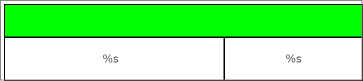
VISUALIZATION VISU_ETAPE_REGEN  // 363x81
VAR_IN_OUT
	COM: BLOCK_RS232_ONBOARD_V4;
END_VAR
    Textfield (4,37 220x44), "%s", text list: 'TextList_CryoPump', text index: COM.STEP_REGEN_ID
    Rectangle (4,4 359x33), colour toggle: COM.STATE_Regen, text list: 'TextList_CryoPump', text index: 43
    Textfield (224,37 139x44), "%s", text variable: COM.VAR_Affichage, text list: 'TextList_CryoPump', text index: COM.ID_ERREUR_REGEN
    Rectangle (4,4 359x33), colour toggle: COM.STATE_Regen, invisible if: not(COM.Regen_completed), text list: 'TextList_CryoPump', text index: 43
END_VISUALIZATION

(* stored: Version 1.1.0.1, ProductVersion 3.1.4026.18
   Visu VISU_ETAPE_REGEN: Id {ee4d141a-0400-47f9-9301-9bb3fb401d96} *)
